Universal Robots PolyScope program: forceUr3e_v0.urp

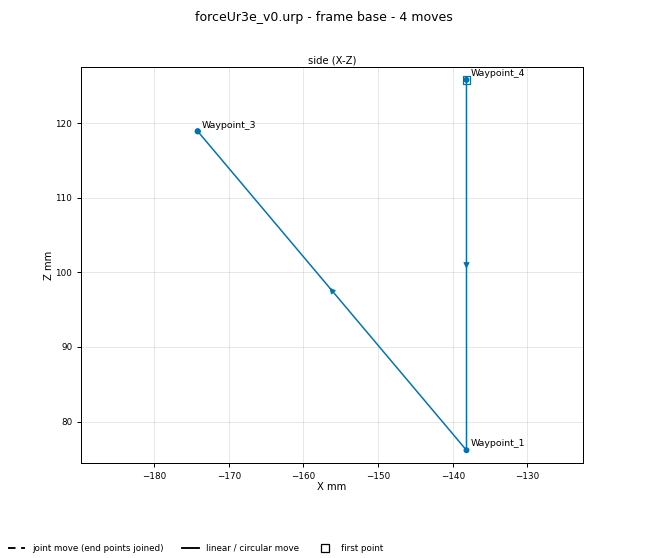
[picture p0: tool path of forceUr3e_v0.urp in frame base, 4 of 4 moves have a stored position in this frame; points joined in program order, loops and branches not executed]
Program forceUr3e_v0 (installation=cb directory=/programs/usbdisk createdIn=5.3.0.64176 lastSavedIn=5.9.3.1031212 robotSerialNumber=20205300403)
Calibrated DH parameters: a=[-0.000043, -0.226611, -0.210721, 0.000054, -0.000126, 0]; d=[0.151936, -135.571411, 139.543118, -3.840954, 0.085412, 0.092221]; alpha=[1.570659, 0.000657, 0.008441, 1.573113, -1.573724, 0]; deltaTheta=[0, -0.374636, 0.5324, -0.157775, 0.000002, 0.000001]
Robot Program (runOnlyOnce=false)
  var_send := False
  fuerza := [0,0,2,0,0,0]
  vel := [0.1,0.1,1,0.17,0.17,0.17]
  vel_2 := [0.01,0.01,3,0.0017,0.17,0.17]
  sel := [0,0,1,0,0,0]
  open := socket_open("158.42.58.182",5000)
  Script: socket_send_string("get")
  Script: textmsg("conexion establecida")
  Script: force_mode_set_damping(0.05)
  Script: force_mode_set_gain_scaling(2)
  MoveL speed 250 mm/s, acceleration 1200 mm/s^2 (useActiveTCP=true) feature=Base
    Wait Sleep waitTime=0.1
    var_send := True
    Script: zero_ftsensor()
    Wait Sleep waitTime=0.2
    Waypoint Waypoint_4: motionParameters(jointSpeed=1.047198 jointAcceleration=1.396263 cartesianSpeed=0.05 cartesianAcceleration=1.2); TCP in base x=-138.162 y=-295.668 z=125.787 mm, rx=2.4622 ry=1.9512 rz=0 rad; joints [-91.448, -91.406, -101.819, -76.603, 90.505, 101.897] deg; TCP offset x=0 y=0 z=130 mm, rx=0 ry=0 rz=0 rad
    Script: force_mode(Joint_6_name,sel,fuerza,2,vel_2)
    Waypoint Waypoint_1: motionParameters(jointSpeed=1.047198 jointAcceleration=1.396263 cartesianSpeed=0.01 cartesianAcceleration=1.2); TCP in base x=-138.157 y=-295.656 z=76.153 mm, rx=-2.4622 ry=-1.9511 rz=0 rad; joints [-91.478, -95.566, -111.57, -62.698, 90.484, 101.982] deg
    Wait Sleep waitTime=0.6
    Waypoint Waypoint_3: motionParameters(jointSpeed=1.047198 jointAcceleration=1.396263 cartesianSpeed=0.2 cartesianAcceleration=1.2); TCP in base x=-174.176 y=-295.618 z=118.893 mm, rx=-2.4622 ry=-1.951 rz=-0.0001 rad; joints [-98.127, -96.033, -98.743, -75.064, 90.503, 95.238] deg
    Wait Sleep waitTime=0.6
    Script: end_force_mode()
    SuppressedNode
      Halt
  SuppressedNode
    Halt
  MoveJ speed 60 deg/s, acceleration 80 deg/s^2 (useActiveTCP=true) feature=Base
    SuppressedNode
      Script: force_mode(Joint_6_name,sel,[0,0,0,0,0,0],2,vel_2)
    Waypoint Waypoint_3: motionParameters(jointSpeed=1.047198 jointAcceleration=1.396263 cartesianSpeed=0.25 cartesianAcceleration=1.2); TCP in base x=-174.176 y=-295.618 z=118.893 mm, rx=-2.4622 ry=-1.951 rz=-0.0001 rad; joints [-98.127, -96.033, -98.743, -75.064, 90.503, 95.238] deg
    Wait Sleep waitTime=2
    Script: end_force_mode()
    SuppressedNode
      Waypoint Waypoint_5: TCP in base x=-341.878 y=-456.011 z=-121.739 mm, rx=-2.2176 ry=-2.1966 rz=-0.0166 rad; joints [40.05, -48.247, 111.709, -152.869, 268.877, 40.787] deg; TCP offset x=0 y=0 z=150 mm, rx=0 ry=0 rz=0 rad
    SuppressedNode
      Wait Sleep waitTime=2
    SuppressedNode
      Waypoint Waypoint_4: TCP in base x=-278.652 y=-540.236 z=-137.821 mm, rx=-2.2176 ry=-2.1966 rz=-0.0166 rad; joints [50.394, -43.648, 104.612, -150.162, 268.975, 51.13] deg
    SuppressedNode
      Halt
  SuppressedNode
    MoveL speed 250 mm/s, acceleration 1200 mm/s^2 (useActiveTCP=true) feature=Base
      Waypoint Waypoint_5: TCP in base x=-181.054 y=-657.099 z=-51.466 mm, rx=-1.8162 ry=-1.8034 rz=-0.6694 rad; joints [67.917, -26.018, 50.783, -76.148, 255.977, 73.403] deg; TCP offset x=0 y=0 z=130 mm, rx=0 ry=0 rz=0 rad
      var_send := False
      Waypoint Waypoint_4: TCP in base x=-138.162 y=-295.668 z=125.787 mm, rx=2.4622 ry=1.9512 rz=0 rad; joints [-91.448, -91.406, -101.819, -76.603, 90.505, 101.897] deg
      Halt
Thread Thread_1 (runOnlyOnce=false)
  var_2 := force()
  var_1 := get_tcp_force()
  var_3 := norm(get_target_tcp_speed())
  var_4 := get_steptime()
  SuppressedNode
    Wait Sleep waitTime=0.1
  If var_send≟ True
    Script: socket_send_string(var_1)
    Script: socket_send_string(var_2)
    Script: socket_send_string("]")
    Script: socket_send_string(var_3)
    SuppressedNode
      Script: socket_send_string("]")
    SuppressedNode
      Script: socket_send_string(var_4)
  Else 
    SuppressedNode
      Script: socket_send_string("a")
  SuppressedNode
    Script: socket_send_string(var_1)
  SuppressedNode
    Script: socket_send_string("a")
  Script: sync()
